Staubli VAL3: getFunctionView.pgx

public program getFunctionView(string& x_sName[])
  local string l_sMessage
begin
  //
  // define your message for the
  // function KEY
  //
  // NOTE is an ARRAY[0..7]
  //
  // example:
  // x_sName[1]="DEMO"
  // active the F2 button

  // HERE
  call language:message(l_sMessage,150)
  x_sName[0]=l_sMessage
  // ALIGN
  call language:message(l_sMessage,134)
  x_sName[1]=l_sMessage
  //
  // DISABLE
  //
  // Paste
  x_sName[3]=" "
  // Mark
  x_sName[4]=" "
  // Insert
  x_sName[5]=" "
  // Delete
  x_sName[6]=" "
end
